FUNCTION_BLOCK CoinButtonsComposite (* Composite Function Block Type *)
  (* Standard: 61499-2 *)
  (* Version 0.2, 2003-12-05, JHC, Rockwell Automation, Renamed from NEWCOMPFB. *)
  (* Version 0.1, 2002-01-08, JHC, Rockwell Automation, Added DLY FB as example. *)
  (* Version 0.0, 2000-05-27, JHC, Rockwell Automation *)
  (* Compiler header: package fb.rt.template; *)
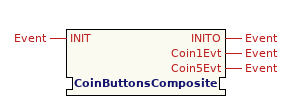
  EVENT_INPUT
    INIT; (* Initialization Request *)
  END_EVENT
  EVENT_OUTPUT
    INITO; (* Initialization Confirm *)
    Coin1Evt;
    Coin5Evt;
  END_EVENT
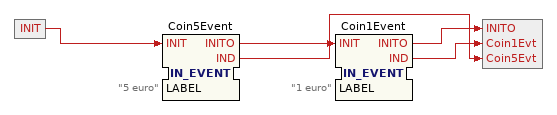
  FBS
    Coin5Event : IN_EVENT(LABEL := "5 euro");
    Coin1Event : IN_EVENT(LABEL := "1 euro");
  END_FBS
  EVENT_CONNECTIONS
    INIT TO Coin5Event.INIT;
    Coin5Event.INITO TO Coin1Event.INIT;
    Coin1Event.INITO TO INITO;
    Coin5Event.IND TO Coin5Evt;
    Coin1Event.IND TO Coin1Evt;
  END_CONNECTIONS
END_FUNCTION_BLOCK
